FUNCTION_BLOCK WorkpieceSensor (* Message Exchange example (slide 47): WPSensor / a1WPS1 - requests the cylinder's round trip service when a workpiece arrives *)
  (* Standard: 61499-2; Description: Copyright (c) 2026 Meisterschulen am Ostbahnhof This program and the accompanying materials are made available under the terms of the Eclipse Public License 2.0 which is available at https://www.eclipse.org/legal/epl-2.0/ SPDX-License-Identifier: EPL-2.0 *)
  (* Version 1.0, 2026-09-03, Franz Höpfinger, Meisterschulen am Ostbahnhof, SoA implementation in function blocks (IEC 61499 primer course, Module 6, Valeriy Vyatkin, slide 47), WPSensor/a1WPS1 role: uses EVENT_HS_ACK_WSTRING (REQ/CNF only) on its ACTIVATE plug, matching the slide's ACTIVATE>> pin name *)
  PACKAGE Meins::DesingPatterns::HandshakePattern;
  IMPORT Meins::DesingPatterns::HandshakePattern::const::MessageExchangeConst;
  (* Documentation:
  Workpiece-arrival sensor (WPSensor/a1WPS1 in the "SoA implementation in function blocks" diagram, IEC 61499 primer course, Module 6, Valeriy Vyatkin, slide 47) - one of the four function blocks in the CylH message-exchange example (slides 42-46 for the message sequence chart this reconstructs).
   Uses EVENT_HS_ACK_WSTRING as a Plug named ACTIVATE (matching the slide's ACTIVATE>> pin): on DETECT (the simulated sensor firing - fire it manually in FORTE monitoring to drive the demo) it sends REQ carrying MessageExchangeConst::REQ_TRIP ("trip", matching the MSC's REQ,"trip"); reports DONE once the matching CNF (expected payload RSP_CYL_TRIP_COMPLETE) comes back from CylinderOrchestrator.
   In the real MSC (slides 42-46) this role is split between two lifelines, WPS (reports its own arrival, RSP,"WPS,1") and MES (decides to request the trip, REQ,"trip"); the FB diagram on slide 47 merges both into this single WPSensor block with one ACTIVATE connection straight into the orchestrator - followed here 1:1.
   See HandshakePattern.md in this folder, section "Die Quelle der 'push,100'-Notation", for the full write-up and the other three function blocks of this example (DropSinkService, CylinderOrchestrator, CylinderService).
  *)
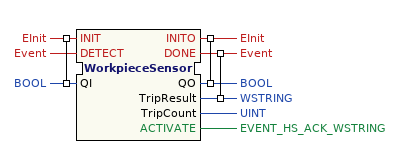
  EVENT_INPUT
    INIT : EInit WITH QI; (* Initialization Request *)
    DETECT; (* Simulated sensor trigger: a workpiece has arrived at the designated place *)
  END_EVENT
  EVENT_OUTPUT
    INITO : EInit WITH QO; (* Initialization Confirm *)
    DONE WITH TripResult; (* The round trip was confirmed complete *)
  END_EVENT
  VAR_INPUT
    QI : BOOL; (* Input event qualifier *)
  END_VAR
  VAR_OUTPUT
    QO : BOOL; (* Output event qualifier *)
    TripResult : WSTRING; (* Payload of the last received CNF (expected: MessageExchangeConst::RSP_CYL_TRIP_COMPLETE) *)
    TripCount : UINT; (* Number of completed round trips (demo counter) *)
  END_VAR
  PLUGS
    ACTIVATE : adapter::types::bidirectional::Handshake::EVENT_HS_ACK_WSTRING; (* Service plug: sends REQ (+REQD) requesting the round trip, receives CNF (+CNFD) when it completes *)
  END_PLUGS
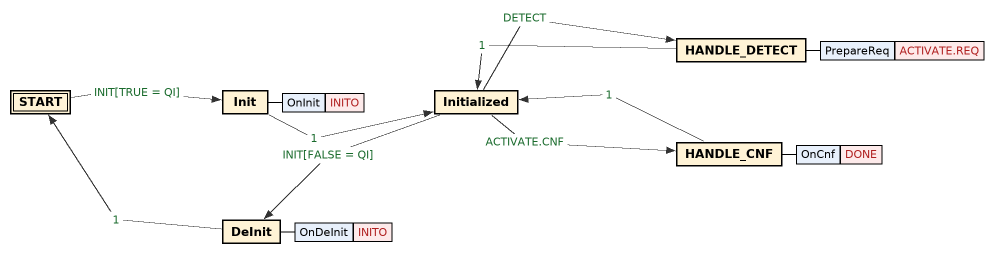
  EC_STATES
    START; (* Uninitialized *)
    Init : OnInit -> INITO; (* Initialization *)
    Initialized; (* Idle, ready to react *)
    DeInit : OnDeInit -> INITO; (* De-initialization *)
    HANDLE_DETECT : PrepareReq -> ACTIVATE.REQ; (* Workpiece arrived: request the round trip *)
    HANDLE_CNF : OnCnf -> DONE; (* Round trip confirmed complete *)
  END_STATES
  EC_TRANSITIONS
    START TO Init := INIT[TRUE = QI];
    Init TO Initialized := 1;
    Initialized TO DeInit := INIT[FALSE = QI];
    DeInit TO START := 1;
    Initialized TO HANDLE_DETECT := DETECT;
    HANDLE_DETECT TO Initialized := 1;
    Initialized TO HANDLE_CNF := ACTIVATE.CNF;
    HANDLE_CNF TO Initialized := 1;
  END_TRANSITIONS
  ALGORITHM OnInit IN ST: (* Reset demo counters/payloads *)
TripResult := "";
TripCount := 0;
QO := QI;
  END_ALGORITHM
  ALGORITHM OnDeInit IN ST: (* De-initialize *)
QO := FALSE;
  END_ALGORITHM
  ALGORITHM PrepareReq IN ST: (* Load REQD with the round-trip request before ACTIVATE.REQ fires *)
ACTIVATE.REQD := MessageExchangeConst::REQ_TRIP;
  END_ALGORITHM
  ALGORITHM OnCnf IN ST: (* Read CNFD, count a completed round trip *)
TripResult := ACTIVATE.CNFD;
TripCount := TripCount + 1;
  END_ALGORITHM
END_FUNCTION_BLOCK
